(*
SPDX-FileCopyrightText: Â© 2026 Oleksandr Tiutyk <trofimich@gmail.com>
SPDX-License-Identifier: MIT
License: https://opensource.org/license/mit
*)

(*!
<summary>Represents an automation component with configurable simulation mode.</summary>
*)

INTERFACE IConfigurableSimulatable EXTENDS ISimulatable

(*!
<summary>Sets whether simulation mode is enabled for the component.</summary>
<param name="value">TRUE to enable simulation mode, FALSE to use physical hardware.</param>
*)
METHOD SetSimulationMode
VAR_INPUT
	value : BOOL;
END_VAR
END_METHOD

END_INTERFACE

(* stored: Version 1.1.0.1
   Itf IConfigurableSimulatable: Id {3effb189-bda6-4e90-acdc-0316c3a2a295}
   Method SetSimulationMode: Id {2ec04501-b180-403d-934c-f7710f1907a0} *)
